PROGRAM FB_Prawidlo
VAR
			//internals
			
			i_seq :INT;
			Czas :ARRAY[0..100] OF TON;
			wyzwolenie         :R_TRIG;
END_VAR

VAR_INPUT			
			//in
			b_Start AT %I* :BOOL;
			b_Stop AT %I* :BOOL;
			bKon_Hamulec1 AT%I* :BOOL	; //kontraktron hamulec 1
			bKon_Hamulec2 AT%I* :BOOL	; //kontraktron hamulec 2
			bKonPodajnik1 AT%I* :BOOL	; //kontraktron podajnik 1
			bKonPodajnik2 AT%I* :BOOL	; //kontraktron podajnik 2
			bCzHamulec AT%I* :BOOL	; //czujnik hamulec 
			bZaladowany AT%I* :BOOL	; //czujnik hamulec 
END_VAR
 //OUT	
VAR_OUTPUT

			 bZaworPodnosnik1 AT%Q* :BOOL	;	// cewka podnośnik 1
			 bZaworPodnosnik2 AT%Q* :BOOL	;	// cewka podnośnik 2
			 bZaworHamulec AT%Q* :BOOL	;	// cewka hamulec
	 		 bZgodaNaRuch AT%Q* :BOOL	;	// cewka hamulec
			 bLaduj AT%Q* :BOOL	;	// czeka na ladunek 
END_VAR

CASE i_seq OF 
	
0:(*inicjalizacja i info o starcie *)


	bZaworPodnosnik1	:=TRUE;
	bZaworPodnosnik2	:=FALSE;
	bZaworHamulec		:=FALSE;
	bZgodaNaRuch 		:=FALSE;
	bLaduj				:=FALSE;
		 
		 IF b_Start=TRUE  THEN
		
		 
		 i_seq:=5;
		 
		END_IF

5:(*jeśli start to podnieś prawidlo do gory wystaw bita że można wydać pudełko  *)

		
			 bZgodaNaRuch		:=TRUE;
			 bZaworHamulec		:=TRUE;
			 
		 IF bKon_Hamulec1=TRUE THEN	 
			 i_seq:=10;
		 END_IF
		 
10:(*jeśli zgoda na ruch to czeka na czujnik  *)	 

	IF Czas[0].Q=TRUE THEN
		
		bZaworPodnosnik1	:=FALSE;
		bZaworPodnosnik2	:=TRUE;
	
		i_seq:=15;
	
	
	END_IF

15:(*czeka na załadunek *)	 

	IF bKonPodajnik1=TRUE THEN
		
	
		bLaduj				:=TRUE;
		i_seq:=20;
	END_IF

20:(*zaladowywuje *)	 

	IF wyzwolenie.Q=TRUE THEN
		bZaworPodnosnik1	:=TRUE;
		bZaworPodnosnik2	:=FALSE;
	i_seq:=25;
	
	END_IF
25:(*zwalnia hamulec i wraca do punktu wyjścia  *)

	IF czas[1].Q=TRUE THEN
	bZaworHamulec		:=FALSE;	
	bLaduj				:=FALSE;
	i_seq:=30;		
	
	END_IF
	
30:

	IF czas[2].Q=TRUE AND bCzHamulec=FALSE  THEN

	i_seq:=5;	
	
	END_IF

	
	

END_CASE

Czas[0](IN:=bCzHamulec, PT:=T#200MS);
Czas[1](IN:=i_seq=25, PT:=T#1S);
Czas[2](IN:=i_seq=30, PT:=T#2S);

		IF b_Stop=TRUE THEN
			
		i_seq:=0;
		
		END_IF
		wyzwolenie(CLK:=bZaladowany);

END_PROGRAM

(* stored: Version 1.1.0.1, ProductVersion 3.1.4022.12
   POU FB_Prawidlo: Id {8b2179ba-161d-4516-9526-cc35fecb993d}, SpecialFunc None *)
